INTERFACE I_AsyncResponseSessionData EXTENDS I_SessionData

METHOD PUBLIC Error
VAR_INPUT
	ErrorCode : T_MAXSTRING;
	Message : T_MAXSTRING;
END_VAR
END_METHOD

PROPERTY PUBLIC IsPending : BOOL
GET
END_GET
END_PROPERTY

METHOD PUBLIC Success
VAR_INPUT
END_VAR
END_METHOD

METHOD PUBLIC SuccessWithPayload
VAR_INPUT
	PayloadDataAddress : PVOID;
	PayloadDataSize : UDINT;
END_VAR
END_METHOD

PROPERTY PUBLIC SuggestedRetryDelayInMs : UDINT
GET
END_GET
SET
END_SET
END_PROPERTY

METHOD PUBLIC TryUpdateServerResponse : BOOL
VAR_INPUT
	Response : I_ServerResponse;
END_VAR
END_METHOD

END_INTERFACE

(* stored: Version 1.1.0.1, ProductVersion 3.1.4024.15
   Itf I_AsyncResponseSessionData: Id {a08a9dea-a80a-0ef0-0fd9-859e178535e4}
   Method Error: Id {e455a056-627c-0b2c-0610-56ca0c23ea4a}
   Property IsPending: Id {16f74dd1-5793-0c40-090c-6134363ac5b1}
   Get Get: Id {a34b0d10-5c56-0b2d-2495-647bae8e99d1}
   Method Success: Id {75cd3cb1-57be-07d1-219d-964b01e7dc95}
   Method SuccessWithPayload: Id {07315348-1ab1-0d14-1318-d3376dc52dba}
   Property SuggestedRetryDelayInMs: Id {1ada00b3-979f-07a4-1392-5c7c34d98b11}
   Get Get: Id {048adede-699a-06f5-2c28-ba5adca76381}
   Set Set: Id {6dcbd7f2-c809-0bd3-0cce-fc87ad0cfbe4}
   Method TryUpdateServerResponse: Id {b5a26c58-eb42-0a78-205f-c0411c9b0741} *)
